% RSLogix 500 project AnalogTank_ALARMS_NOTIFICATIONS.RSS, saved by version 8.30.00.16 %
PROJECT "UNTITLED"    % processor: Bul.1763 MicroLogix 1100 Series B %

PROGRAM FILES
  LAD 2 "MAIN"  4 rungs
  LAD 3 "IO"  4 rungs
  LAD 4 "CONTROLS"  6 rungs
  LAD 5 "ALARMS"  7 rungs

DATA FILES
  O0 OUTPUT  5 elements
  I1 INPUT  14 elements
  S2 STATUS  66 elements
  B3 BINARY  10 elements
  T4 TIMER  4 elements
  C5 COUNTER  1 elements
  R6 CONTROL  1 elements
  N7 INTEGER  1 elements
  F8 FLOAT  1 elements

LADDER 2 "MAIN"
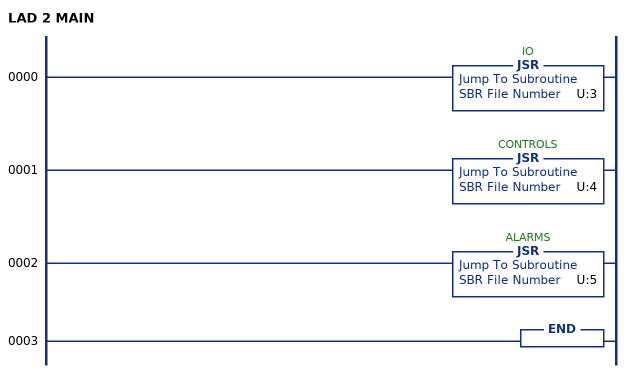
% Rung: 0 %
SOR JSR U:3 EOR
%   U:3  "IO" %
% Rung: 1 %
SOR JSR U:4 EOR
%   U:4  "CONTROLS" %
% Rung: 2 %
SOR JSR U:5 EOR
%   U:5  "ALARMS" %
% Rung: 3 %
SOR END EOR

LADDER 3 "IO"
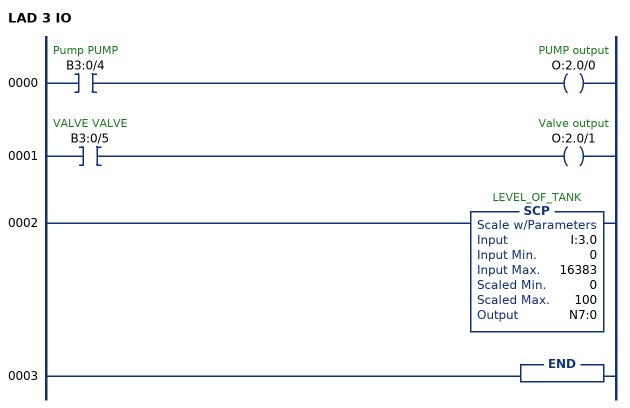
% Rung: 0 %
SOR XIC B3:0/4 OTE O:2.0/0 EOR
%   B3:0/4  PUMP  "Pump" %
%   O:2.0/0  "PUMP output" %
% Rung: 1 %
SOR XIC B3:0/5 OTE O:2.0/1 EOR
%   B3:0/5  VALVE  "VALVE" %
%   O:2.0/1  "Valve output" %
% Rung: 2 %
SOR SCP I:3.0 0 16383 0 100 N7:0 EOR
%   I:3.0  "analog input" %
%   N7:0  LEVEL_OF_TANK %
% Rung: 3 %
SOR END EOR

LADDER 4 "CONTROLS"
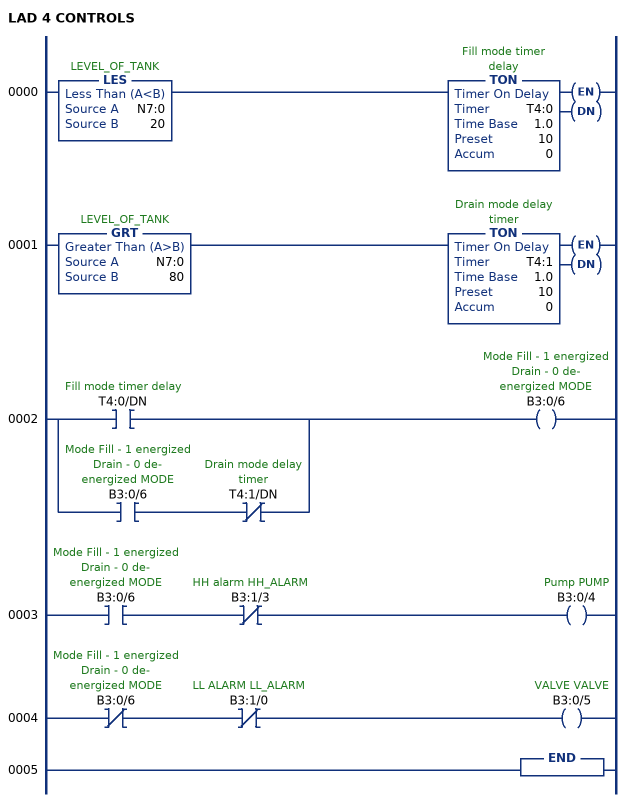
% Rung: 0 %
SOR LES N7:0 20 TON T4:0 1.0 10 0 EOR
%   N7:0  LEVEL_OF_TANK %
%   T4:0  "Fill mode timer delay" %
% Rung: 1 %
SOR GRT N7:0 80 TON T4:1 1.0 10 0 EOR
%   N7:0  LEVEL_OF_TANK %
%   T4:1  "Drain mode delay timer" %
% Rung: 2 %
SOR BST XIC T4:0/DN NXB XIC B3:0/6 XIO T4:1/DN BND OTE B3:0/6 EOR
%   T4:0  "Fill mode timer delay" %
%   B3:0/6  MODE  "Mode Fill - 1 energized Drain - 0 de- energized" %
%   T4:1  "Drain mode delay timer" %
% Rung: 3 %
SOR XIC B3:0/6 XIO B3:1/3 OTE B3:0/4 EOR
%   B3:0/6  MODE  "Mode Fill - 1 energized Drain - 0 de- energized" %
%   B3:1/3  HH_ALARM  "HH alarm" %
%   B3:0/4  PUMP  "Pump" %
% Rung: 4 %
SOR XIO B3:0/6 XIO B3:1/0 OTE B3:0/5 EOR
%   B3:0/6  MODE  "Mode Fill - 1 energized Drain - 0 de- energized" %
%   B3:1/0  LL_ALARM  "LL ALARM" %
%   B3:0/5  VALVE  "VALVE" %
% Rung: 5 %
SOR END EOR

LADDER 5 "ALARMS"
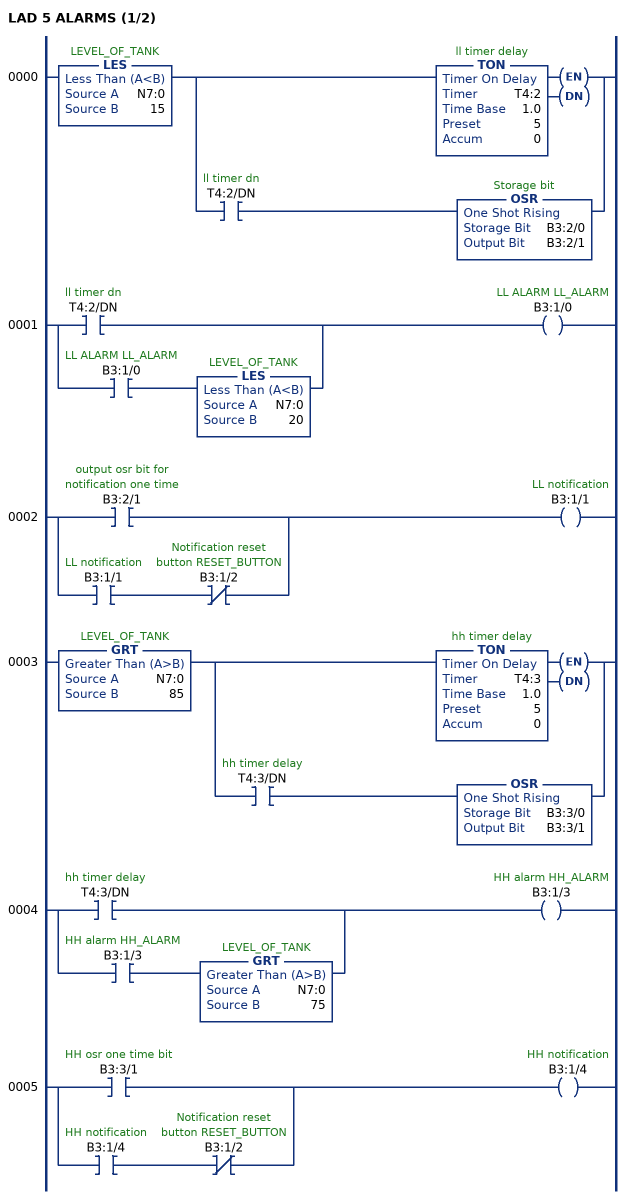
% Rung: 0 %
SOR LES N7:0 15 BST TON T4:2 1.0 5 0 NXB XIC T4:2/DN OSR B3:2/0 B3:2/1 BND EOR
%   N7:0  LEVEL_OF_TANK %
%   T4:2  "ll timer delay" %
%   T4:2/DN  "ll timer dn" %
%   B3:2/0  "Storage bit" %
%   B3:2/1  "output osr bit for notification one time" %
% Rung: 1 %
SOR BST XIC T4:2/DN NXB XIC B3:1/0 LES N7:0 20 BND OTE B3:1/0 EOR
%   T4:2/DN  "ll timer dn" %
%   B3:1/0  LL_ALARM  "LL ALARM" %
%   N7:0  LEVEL_OF_TANK %
% Rung: 2 %
SOR BST XIC B3:2/1 NXB XIC B3:1/1 XIO B3:1/2 BND OTE B3:1/1 EOR
%   B3:2/1  "output osr bit for notification one time" %
%   B3:1/1  "LL notification" %
%   B3:1/2  RESET_BUTTON  "Notification reset button" %
% Rung: 3 %
SOR GRT N7:0 85 BST TON T4:3 1.0 5 0 NXB XIC T4:3/DN OSR B3:3/0 B3:3/1 BND EOR
%   N7:0  LEVEL_OF_TANK %
%   T4:3  "hh timer delay" %
%   B3:3/1  "HH osr one time bit" %
% Rung: 4 %
SOR BST XIC T4:3/DN NXB XIC B3:1/3 GRT N7:0 75 BND OTE B3:1/3 EOR
%   T4:3  "hh timer delay" %
%   B3:1/3  HH_ALARM  "HH alarm" %
%   N7:0  LEVEL_OF_TANK %
% Rung: 5 %
SOR BST XIC B3:3/1 NXB XIC B3:1/4 XIO B3:1/2 BND OTE B3:1/4 EOR
%   B3:3/1  "HH osr one time bit" %
%   B3:1/4  "HH notification" %
%   B3:1/2  RESET_BUTTON  "Notification reset button" %

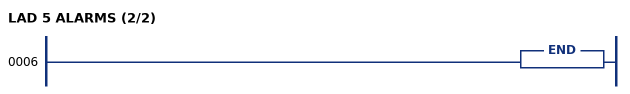
% Rung: 6 %
SOR END EOR

OTHER DOCUMENTED ADDRESSES
  ALARM  "Alarm BIT"
  B3:0/0  LL_SWITCH  "LL Swicth"
  B3:0/1  L_SWITCH  "L Switch"
  B3:0/2  H_SWITCH  "H Switch"
  B3:0/3  HH_SWITCH  "HH Switch"
  I:1.0/0  "LL switch input"
  I:1.0/1  "L switch input"
  I:1.0/2  "H Switch input"
  I:1.0/3  "HH switch input"

DATA TABLE (non-zero values as saved)
DATA T4
% .PRE .ACC %
% T4:0 % 10 0
% T4:1 % 10 0
% T4:2 % 5 0
% T4:3 % 5 0
